// TIA Portal V20 export
DATA_BLOCK "ControlNodes"   // DB51
// stored: MemoryReserve 100, Namespace Unit1.Em6
   VAR
      em : "LAF_typeEmControlNode";
      emstate { S7_SetPoint := 'True'} : "LUC_typeStates";
      cm { S7_SetPoint := 'True'} : "Unit1.Em6.typeCmControlNode";
      citiMap : Struct
         PMC : "LER_PMC_Input_Data";
         FlexNet { S7_SetPoint := 'True'} : "LER_FlexNet_Data";
      END_STRUCT;
      hotPressLeft : "Unit1.Em6.typeSequenceControlNode";
      emData : "Unit1.Em6.typeEmDataControlNode";
      SpecialFunctionMode : Struct
         DryRun : Struct
            JRdetectPV : Array[0..15] of Bool;
         END_STRUCT;
      END_STRUCT;
      cmHotpressLeftSafetyPin : "LBC_typeDigitalSignalControlNode";
      cmHotpressLeftJRDetect : "LBC_typeDigitalSignalControlNode";
      cmHotpressLeftStageLiftFrontUpDown : "LBC_typeTwoWayActuatorControlNode";
      cmHotpressLeftStageLiftRearUpDown : "LBC_typeTwoWayActuatorControlNode";
      cmHotpressLeftStageLiftAllUpDown : "LBC_typeTwoWayActuatorControlNode";
      cmHotPressLeftServoPress : "LER_typeServoPressControlNode";
      cmHotPressLeftTemperature : "LER_typeHeaterControlNode";
   END_VAR
BEGIN
END_DATA_BLOCK
